FUNCTION Convert_TOD_TO_DINT : Hresult
VAR_INPUT
	in : TOD;
	out : REFERENCE TO DINT;
END_VAR
VAR
	converted : DINT;
END_VAR

converted := TOD_TO_DINT(in);

IF (DINT_TO_TOD(converted) <> in) THEN
	Convert_TOD_TO_DINT := INCOMPATIBLE;
	RETURN;
END_IF

out := converted;

END_FUNCTION

(* stored: Version 1.1.0.1, ProductVersion 3.1.4024.12
   POU Convert_TOD_TO_DINT: Id {71a43749-9b5e-429d-aa25-14c3b0a0755e}, SpecialFunc None *)
